TYPE DUT1 :
STRUCT
	i : INT;
	j : REAL;
	b : BOOL;
	
END_STRUCT
END_TYPE

(* stored: Version 1.1.0.1, ProductVersion 3.1.4024.12
   DUT DUT1: Id {b29aa91d-b109-4bef-834d-9919a93aa820} *)
